TYPE ASCF_CC_OPCUACS_ScheduleDataType2 :
STRUCT
	NextID			: INT					:= 1;
	Schedule		: ARRAY[0..4] OF INT	:= [0, 0, 0, 0, 0];		//war vorher 00000
END_STRUCT
END_TYPE

(* stored: Version 1.1.0.1, ProductVersion 3.1.4026.4
   DUT ASCF_CC_OPCUACS_ScheduleDataType2: Id {d8f7ee2f-5a15-477e-a381-035860f06a63} *)
